SUBAPPLICATION Uebung_010 (* SoftKey_F1 auf DigitalOutput_Q1 *)
  (* Standard: 61499-2 *)
  (* Version 1.0, 2023-10-23, franz *)
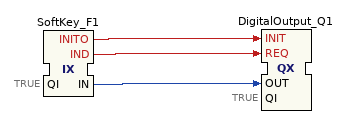
  FBS
    DigitalOutput_Q1 : QX(QI := TRUE);
    SoftKey_F1 : IX(QI := TRUE);
  END_FBS
  EVENT_CONNECTIONS
    SoftKey_F1.INITO TO DigitalOutput_Q1.INIT;
    SoftKey_F1.IND TO DigitalOutput_Q1.REQ;
  END_CONNECTIONS
  DATA_CONNECTIONS
    SoftKey_F1.IN TO DigitalOutput_Q1.OUT;
  END_CONNECTIONS
END_SUBAPPLICATION
